Staubli VAL3: jump.pgx

program jump()
begin
  while true
    movej(jump1,flange,mNomSpeed)
    movej(jump2,flange,mNomSpeed)
    waitEndMove()
  endWhile
end
